(* Logix 5000 project; controller SPONGENT Emulate 5570 rev 30.12; software revision 30.00 *)

TASK MainTask (periodic, rate 500 ms, priority 1, watchdog 500 ms) : MainProgram

MODULES
   Local : Emulate 5570 (ICP 2, rev 30.12)
       : vendor 1 type 0 code 15 (ICP 3, rev 1.1, Output RPI 50 ms)
END_MODULES

VAR_GLOBAL   (* controller tags *)
   SCAN_CYCLE_TIME : DINT := 12;
END_VAR

PROGRAM MainProgram   (* main routine MainRoutine *)
VAR
   Spon_Absorb_i : DINT := 1;
   Spon_BAD_HASHBITLEN : DINT;
   Spon_capacity : DINT := 80;
   Spon_Check_i : DINT := 11;
   Spon_Check_j : DINT := 11;
   Spon_Digest : DINT[256] := ([0] := 211, [1] := 187, [2] := 154, [3] := 14, [4] := 13, [5] := 90, [6] := 242, [7] := 217, [8] := 117, [9] := 72, [10] := 177);
   Spon_DIGESTSIZE : DINT := 88;
   Spon_Hash_i : DINT := 1;
   Spon_Hash_index : DINT;
   Spon_Hash_statrIndex : DINT := 10;
   Spon_hashbitlen : DINT := 88;
   Spon_i : DINT;
   Spon_INV_IV : DINT[512] := ([0] := 63488);
   Spon_IV : DINT[512] := ([0] := 63);
   Spon_j : DINT;
   Spon_Message : DINT[1024] := ([0] := 48, [1] := 48, [2] := 48, [3] := 48, [4] := 48, [5] := 48, [6] := 48, [7] := 48, [8] := 48, [9] := 48, [10] := 48, [11] := 48, [12] := 48, [13] := 48, [14] := 48, [15] := 48, [16] := 48, [17] := 48, [18] := 48, [19] := 48, [20] := 48, [21] := 48, [22] := 48, [23] := 48, [24] := 48, [25] := 48, [26] := 48);
   Spon_messageblock : DINT[1024] := ([0] := 72);
   Spon_MsgBitLen : DINT;
   Spon_nBits : DINT := 88;
   Spon_nRounds : DINT := 45;
   Spon_nSBox : DINT := 11;
   Spon_Pad_bitpos : DINT;
   Spon_Pad_byteind : DINT := 1;
   Spon_Pad_indx : DINT;
   Spon_Permute_i : DINT := 45;
   Spon_Permute_j : DINT := 11;
   Spon_Player_i : DINT := 11;
   Spon_Player_j : DINT := 8;
   Spon_Player_PermutedBitNo : DINT := 87;
   Spon_Player_pos : DINT := 7;
   Spon_Player_tmp : DINT;
   Spon_Player_x : DINT;
   Spon_Player_y : DINT := 10;
   Spon_Player_z : DINT := 87;
   Spon_R_SizeInBytes : DINT := 1;
   Spon_rate : DINT := 8;
   Spon_remainingbitlen : DINT;
   Spon_res : DINT;
   Spon_retnuoCl_lfsr : DINT := 63488;
   Spon_retnuoCl_res : DINT;
   Spon_S : DINT[16] := ([0] := 14, [1] := 13, [2] := 11, [4] := 2, [5] := 1, [6] := 4, [7] := 15, [8] := 7, [9] := 10, [10] := 8, [11] := 5, [12] := 9, [13] := 12, [14] := 3, [15] := 6);
   Spon_SBoxLayer : DINT[256] := ([0] := 238, [1] := 237, [2] := 235, [3] := 224, [4] := 226, [5] := 225, [6] := 228, [7] := 239, [8] := 231, [9] := 234, [10] := 232, [11] := 229, [12] := 233, [13] := 236, [14] := 227, [15] := 230, [16] := 222, [17] := 221, [18] := 219, [19] := 208, [20] := 210, [21] := 209, [22] := 212, [23] := 223, [24] := 215, [25] := 218, [26] := 216, [27] := 213, [28] := 217, [29] := 220, [30] := 211, [31] := 214, [32] := 190, [33] := 189, [34] := 187, [35] := 176, [36] := 178, [37] := 177, [38] := 180, [39] := 191, [40] := 183, [41] := 186, [42] := 184, [43] := 181, [44] := 185, [45] := 188, [46] := 179, [47] := 182, [48] := 14, [49] := 13, [50] := 11, [52] := 2, [53] := 1, [54] := 4, [55] := 15, [56] := 7, [57] := 10, [58] := 8, [59] := 5, [60] := 9,
        [61] := 12, [62] := 3, [63] := 6, [64] := 46, [65] := 45, [66] := 43, [67] := 32, [68] := 34, [69] := 33, [70] := 36, [71] := 47, [72] := 39, [73] := 42, [74] := 40, [75] := 37, [76] := 41, [77] := 44, [78] := 35, [79] := 38, [80] := 30, [81] := 29, [82] := 27, [83] := 16, [84] := 18, [85] := 17, [86] := 20, [87] := 31, [88] := 23, [89] := 26, [90] := 24, [91] := 21, [92] := 25, [93] := 28, [94] := 19, [95] := 22, [96] := 78, [97] := 77, [98] := 75, [99] := 64, [100] := 66, [101] := 65, [102] := 68, [103] := 79, [104] := 71, [105] := 74, [106] := 72, [107] := 69, [108] := 73, [109] := 76, [110] := 67, [111] := 70, [112] := 254, [113] := 253, [114] := 251, [115] := 240, [116] := 242, [117] := 241, [118] := 244, [119] := 255, [120] := 247,
        [121] := 250, [122] := 248, [123] := 245, [124] := 249, [125] := 252, [126] := 243, [127] := 246, [128] := 126, [129] := 125, [130] := 123, [131] := 112, [132] := 114, [133] := 113, [134] := 116, [135] := 127, [136] := 119, [137] := 122, [138] := 120, [139] := 117, [140] := 121, [141] := 124, [142] := 115, [143] := 118, [144] := 174, [145] := 173, [146] := 171, [147] := 160, [148] := 162, [149] := 161, [150] := 164, [151] := 175, [152] := 167, [153] := 170, [154] := 168, [155] := 165, [156] := 169, [157] := 172, [158] := 163, [159] := 166, [160] := 142, [161] := 141, [162] := 139, [163] := 128, [164] := 130, [165] := 129, [166] := 132, [167] := 143, [168] := 135, [169] := 138, [170] := 136, [171] := 133, [172] := 137, [173] := 140, [174] := 131, [175] := 134, [176] := 94, [177] := 93, [178] := 91, [179] := 80, [180] := 82,
        [181] := 81, [182] := 84, [183] := 95, [184] := 87, [185] := 90, [186] := 88, [187] := 85, [188] := 89, [189] := 92, [190] := 83, [191] := 86, [192] := 158, [193] := 157, [194] := 155, [195] := 144, [196] := 146, [197] := 145, [198] := 148, [199] := 159, [200] := 151, [201] := 154, [202] := 152, [203] := 149, [204] := 153, [205] := 156, [206] := 147, [207] := 150, [208] := 206, [209] := 205, [210] := 203, [211] := 192, [212] := 194, [213] := 193, [214] := 196, [215] := 207, [216] := 199, [217] := 202, [218] := 200, [219] := 197, [220] := 201, [221] := 204, [222] := 195, [223] := 198, [224] := 62, [225] := 61, [226] := 59, [227] := 48, [228] := 50, [229] := 49, [230] := 52, [231] := 63, [232] := 55, [233] := 58, [234] := 56, [235] := 53, [236] := 57, [237] := 60, [238] := 51, [239] := 54, [240] := 110,
        [241] := 109, [242] := 107, [243] := 96, [244] := 98, [245] := 97, [246] := 100, [247] := 111, [248] := 103, [249] := 106, [250] := 104, [251] := 101, [252] := 105, [253] := 108, [254] := 99, [255] := 102);
   Spon_Slayer_input : DINT := 241;
   Spon_Slayer_res : DINT;
   Spon_Squeeze_i : DINT := 1;
   Spon_State : DINT[256] := ([0] := 177, [1] := 249, [2] := 148, [3] := 195, [4] := 111, [5] := 169, [6] := 251, [7] := 236, [8] := 167, [9] := 175, [10] := 126);
   Spon_State_tmp : DINT[256] := ([0] := 177, [1] := 249, [2] := 148, [3] := 195, [4] := 111, [5] := 169, [6] := 251, [7] := 236, [8] := 167, [9] := 175, [10] := 126);
   Spon_SUCCESS : DINT;
   Spon_Ver : DINT := 88808;
   Test_i : DINT := 27;
END_VAR

ROUTINE MainRoutine   (* ladder *)
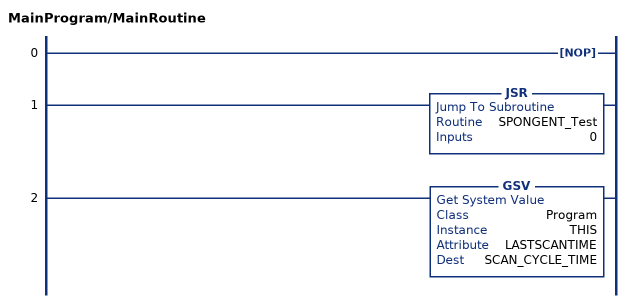
   0: NOP();
   1: JSR(SPONGENT_Test,0);
   2: GSV(Program,THIS,LASTSCANTIME,SCAN_CYCLE_TIME);
END_ROUTINE

ROUTINE SPONGENT   (* structured text *)
   JSR(SPONGENT_Init);
   
   
   
   //Spon_hashval, state
   
   
   
   
   /* Absorb available message blocks */
   Spon_Hash_statrIndex:=0;
   While Spon_MsgBitLen >= Spon_rate do
   	//memcpy(state.messageblock, data, R_SizeInBytes);
   	for Spon_Hash_i:=0 to Spon_R_SizeInBytes-1 by 1 do
   		Spon_messageblock[Spon_Hash_i]:=Spon_Message[Spon_Hash_statrIndex+Spon_Hash_i];
   	end_for;
   
   
   	JSR(SPONGENT_Absorb);
   	Spon_MsgBitLen:=Spon_MsgBitLen-Spon_rate;
   	Spon_Hash_statrIndex:=Spon_Hash_statrIndex+Spon_R_SizeInBytes;
   
   end_while;
   
   
   
   //databitlen/8 + (databitlen%8?1:0)
   Spon_Hash_index:=Spon_MsgBitLen mod 8;
   if Spon_Hash_index=0 then
   	Spon_Hash_index:=Spon_MsgBitLen / 8;
   else
   	Spon_Hash_index:=Spon_MsgBitLen / 8 + 1;
   end_if;
   
   if Spon_MsgBitLen>0 then
   //memcpy(state.messageblock, data, databitlen/8 + (databitlen%8?1:0));
   	for Spon_Hash_i:=0 to Spon_Hash_index-1 by 1 do
   		Spon_messageblock[Spon_Hash_i]:=Spon_Message[Spon_Hash_statrIndex+Spon_Hash_i];
   	end_for;
   	Spon_remainingbitlen:=Spon_MsgBitLen;
   else
   	for Spon_Hash_i:=0 to Spon_R_SizeInBytes-1 by 1 do
   		Spon_messageblock[Spon_Hash_i]:=0;
   	end_for;
   	Spon_remainingbitlen:=Spon_MsgBitLen;
   end_if;
   
   
   JSR(SPONGENT_Pad);
   
   JSR(SPONGENT_Absorb);
   Spon_hashbitlen:=Spon_hashbitlen+Spon_rate;
   
   /* Squeeze data blocks */
   Spon_Hash_statrIndex:=0;
   while Spon_hashbitlen<Spon_DIGESTSIZE do
   	JSR(SPONGENT_Squeeze);
   
   
   	for Spon_Hash_i:=0 to Spon_R_SizeInBytes-1 by 1 do
   		Spon_Digest[Spon_Hash_statrIndex+Spon_Hash_i]:=Spon_messageblock[Spon_Hash_i];
   	end_for;
   
   	Spon_hashbitlen:=Spon_hashbitlen+Spon_rate;
   	Spon_Hash_statrIndex:=Spon_Hash_statrIndex+Spon_R_SizeInBytes;
   
   end_while;
   
   
   
   for Spon_Hash_i:=0 to Spon_R_SizeInBytes-1 by 1 do
   	Spon_Digest[Spon_Hash_statrIndex+Spon_Hash_i]:=Spon_State[Spon_Hash_i];
   end_for;
   
   
   
   
   
   
   
   
   
   
   
   
   
END_ROUTINE

ROUTINE SPONGENT_Absorb   (* structured text *)
   (*
   int i;
   	for(i = 0; i < R_SizeInBytes; i++)
   		state->value[i] ^= state->messageblock[i];
    	Permute(state);
   
   	return SUCCESS;
   
   	*)
   
   For Spon_Absorb_i:=0 to Spon_R_SizeInBytes-1 by 1 Do
   	Spon_State[Spon_Absorb_i]:= Spon_State[Spon_Absorb_i] Xor Spon_messageblock[Spon_Absorb_i];
   End_for;
   
   JSR(SPONGENT_Permute);
END_ROUTINE

ROUTINE SPONGENT_Init   (* structured text *)
   	Spon_INV_IV[0]:=25344;
   	Spon_INV_IV[1]:=22528;
   	Spon_INV_IV[2]:=38400;
   	Spon_INV_IV[3]:=42240;
   	Spon_INV_IV[4]:=26880;
   	Spon_INV_IV[5]:=6656;
   	Spon_INV_IV[6]:=17920;
   	Spon_INV_IV[7]:=37120;
   	Spon_INV_IV[8]:=41984;
   	Spon_INV_IV[9]:=26880;
   	Spon_INV_IV[10]:=6656;
   	Spon_INV_IV[11]:=17920;
   	Spon_INV_IV[12]:=37120;
   	Spon_INV_IV[13]:=41984;
   	Spon_INV_IV[14]:=26880;
   	Spon_INV_IV[15]:=6656;
   	Spon_INV_IV[16]:=17920;
   	Spon_INV_IV[17]:=37120;
   	Spon_INV_IV[18]:=41984;
   	Spon_INV_IV[19]:=26880;
   	Spon_INV_IV[20]:=6656;
   	Spon_INV_IV[21]:=17920;
   	Spon_INV_IV[22]:=37120;
   	Spon_INV_IV[23]:=41984;
   	Spon_INV_IV[24]:=26880;
   	Spon_INV_IV[25]:=6656;
   	Spon_INV_IV[26]:=17920;
   	Spon_INV_IV[27]:=37120;
   	Spon_INV_IV[28]:=41984;
   	Spon_INV_IV[29]:=26880;
   	Spon_INV_IV[30]:=6656;
   	Spon_INV_IV[31]:=17920;
   	Spon_INV_IV[32]:=37120;
   	Spon_INV_IV[33]:=41984;
   	Spon_INV_IV[34]:=26880;
   	Spon_INV_IV[35]:=6656;
   	Spon_INV_IV[36]:=17920;
   	Spon_INV_IV[37]:=37120;
   	Spon_INV_IV[38]:=41984;
   	Spon_INV_IV[39]:=26880;
   	Spon_INV_IV[40]:=6656;
   	Spon_INV_IV[41]:=17920;
   	Spon_INV_IV[42]:=37120;
   	Spon_INV_IV[43]:=41984;
   	Spon_INV_IV[44]:=26880;
   	Spon_INV_IV[45]:=6656;
   	Spon_INV_IV[46]:=17920;
   	Spon_INV_IV[47]:=37120;
   	Spon_INV_IV[48]:=41984;
   	Spon_INV_IV[49]:=26880;
   	Spon_INV_IV[50]:=6656;
   	Spon_INV_IV[51]:=17920;
   	Spon_INV_IV[52]:=37120;
   	Spon_INV_IV[53]:=41984;
   	Spon_INV_IV[54]:=26880;
   	Spon_INV_IV[55]:=6656;
   	Spon_INV_IV[56]:=17920;
   	Spon_INV_IV[57]:=37120;
   	Spon_INV_IV[58]:=41984;
   	Spon_INV_IV[59]:=26880;
   	Spon_INV_IV[60]:=6656;
   	Spon_INV_IV[61]:=17920;
   	Spon_INV_IV[62]:=37120;
   	Spon_INV_IV[63]:=41984;
   	Spon_INV_IV[64]:=26880;
   	Spon_INV_IV[65]:=6656;
   	Spon_INV_IV[66]:=17920;
   	Spon_INV_IV[67]:=37120;
   	Spon_INV_IV[68]:=41984;
   	Spon_INV_IV[69]:=26880;
   	Spon_INV_IV[70]:=6656;
   	Spon_INV_IV[71]:=17920;
   	Spon_INV_IV[72]:=37120;
   	Spon_INV_IV[73]:=41984;
   	Spon_INV_IV[74]:=26880;
   	Spon_INV_IV[75]:=6656;
   	Spon_INV_IV[76]:=17920;
   	Spon_INV_IV[77]:=37120;
   	Spon_INV_IV[78]:=41984;
   	Spon_INV_IV[79]:=26880;
   	Spon_INV_IV[80]:=6656;
   	Spon_INV_IV[81]:=17920;
   	Spon_INV_IV[82]:=37120;
   	Spon_INV_IV[83]:=41984;
   	Spon_INV_IV[84]:=26880;
   	Spon_INV_IV[85]:=6656;
   	Spon_INV_IV[86]:=17920;
   	Spon_INV_IV[87]:=37120;
   	Spon_INV_IV[88]:=41984;
   	Spon_INV_IV[89]:=26880;
   	Spon_INV_IV[90]:=6656;
   	Spon_INV_IV[91]:=17920;
   	Spon_INV_IV[92]:=37120;
   	Spon_INV_IV[93]:=41984;
   	Spon_INV_IV[94]:=26880;
   	Spon_INV_IV[95]:=6656;
   	Spon_INV_IV[96]:=17920;
   	Spon_INV_IV[97]:=37120;
   	Spon_INV_IV[98]:=41984;
   	Spon_INV_IV[99]:=26880;
   	Spon_INV_IV[100]:=6656;
   	Spon_INV_IV[101]:=17920;
   	Spon_INV_IV[102]:=37120;
   	Spon_INV_IV[103]:=41984;
   	Spon_INV_IV[104]:=26880;
   	Spon_INV_IV[105]:=6656;
   	Spon_INV_IV[106]:=17920;
   	Spon_INV_IV[107]:=37120;
   	Spon_INV_IV[108]:=41984;
   	Spon_INV_IV[109]:=26880;
   	Spon_INV_IV[110]:=6656;
   	Spon_INV_IV[111]:=17920;
   	Spon_INV_IV[112]:=37120;
   	Spon_INV_IV[113]:=41984;
   	Spon_INV_IV[114]:=26880;
   	Spon_INV_IV[115]:=6656;
   	Spon_INV_IV[116]:=17920;
   	Spon_INV_IV[117]:=37120;
   	Spon_INV_IV[118]:=41984;
   	Spon_INV_IV[119]:=26880;
   	Spon_INV_IV[120]:=6656;
   	Spon_INV_IV[121]:=17920;
   	Spon_INV_IV[122]:=37120;
   	Spon_INV_IV[123]:=41984;
   	Spon_INV_IV[124]:=26880;
   	Spon_INV_IV[125]:=6656;
   	Spon_INV_IV[126]:=17920;
   	Spon_INV_IV[127]:=37120;
   	Spon_INV_IV[128]:=41984;
   	Spon_INV_IV[129]:=26880;
   	Spon_INV_IV[130]:=6656;
   	Spon_INV_IV[131]:=17920;
   	Spon_INV_IV[132]:=37120;
   	Spon_INV_IV[133]:=41984;
   	Spon_INV_IV[134]:=26880;
   
   
   	Spon_IV[0]:=198;
   	Spon_IV[1]:=26;
   	Spon_IV[2]:=105;
   	Spon_IV[3]:=165;
   	Spon_IV[4]:=150;
   	Spon_IV[5]:=88;
   	Spon_IV[6]:=98;
   	Spon_IV[7]:=137;
   	Spon_IV[8]:=37;
   	Spon_IV[9]:=150;
   	Spon_IV[10]:=88;
   	Spon_IV[11]:=98;
   	Spon_IV[12]:=137;
   	Spon_IV[13]:=37;
   	Spon_IV[14]:=150;
   	Spon_IV[15]:=88;
   	Spon_IV[16]:=98;
   	Spon_IV[17]:=137;
   	Spon_IV[18]:=37;
   	Spon_IV[19]:=150;
   	Spon_IV[20]:=88;
   	Spon_IV[21]:=98;
   	Spon_IV[22]:=137;
   	Spon_IV[23]:=37;
   	Spon_IV[24]:=150;
   	Spon_IV[25]:=88;
   	Spon_IV[26]:=98;
   	Spon_IV[27]:=137;
   	Spon_IV[28]:=37;
   	Spon_IV[29]:=150;
   	Spon_IV[30]:=88;
   	Spon_IV[31]:=98;
   	Spon_IV[32]:=137;
   	Spon_IV[33]:=37;
   	Spon_IV[34]:=150;
   	Spon_IV[35]:=88;
   	Spon_IV[36]:=98;
   	Spon_IV[37]:=137;
   	Spon_IV[38]:=37;
   	Spon_IV[39]:=150;
   	Spon_IV[40]:=88;
   	Spon_IV[41]:=98;
   	Spon_IV[42]:=137;
   	Spon_IV[43]:=37;
   	Spon_IV[44]:=150;
   	Spon_IV[45]:=88;
   	Spon_IV[46]:=98;
   	Spon_IV[47]:=137;
   	Spon_IV[48]:=37;
   	Spon_IV[49]:=150;
   	Spon_IV[50]:=88;
   	Spon_IV[51]:=98;
   	Spon_IV[52]:=137;
   	Spon_IV[53]:=37;
   	Spon_IV[54]:=150;
   	Spon_IV[55]:=88;
   	Spon_IV[56]:=98;
   	Spon_IV[57]:=137;
   	Spon_IV[58]:=37;
   	Spon_IV[59]:=150;
   	Spon_IV[60]:=88;
   	Spon_IV[61]:=98;
   	Spon_IV[62]:=137;
   	Spon_IV[63]:=37;
   	Spon_IV[64]:=150;
   	Spon_IV[65]:=88;
   	Spon_IV[66]:=98;
   	Spon_IV[67]:=137;
   	Spon_IV[68]:=37;
   	Spon_IV[69]:=150;
   	Spon_IV[70]:=88;
   	Spon_IV[71]:=98;
   	Spon_IV[72]:=137;
   	Spon_IV[73]:=37;
   	Spon_IV[74]:=150;
   	Spon_IV[75]:=88;
   	Spon_IV[76]:=98;
   	Spon_IV[77]:=137;
   	Spon_IV[78]:=37;
   	Spon_IV[79]:=150;
   	Spon_IV[80]:=88;
   	Spon_IV[81]:=98;
   	Spon_IV[82]:=137;
   	Spon_IV[83]:=37;
   	Spon_IV[84]:=150;
   	Spon_IV[85]:=88;
   	Spon_IV[86]:=98;
   	Spon_IV[87]:=137;
   	Spon_IV[88]:=37;
   	Spon_IV[89]:=150;
   	Spon_IV[90]:=88;
   	Spon_IV[91]:=98;
   	Spon_IV[92]:=137;
   	Spon_IV[93]:=37;
   	Spon_IV[94]:=150;
   	Spon_IV[95]:=88;
   	Spon_IV[96]:=98;
   	Spon_IV[97]:=137;
   	Spon_IV[98]:=37;
   	Spon_IV[99]:=150;
   	Spon_IV[100]:=88;
   	Spon_IV[101]:=98;
   	Spon_IV[102]:=137;
   	Spon_IV[103]:=37;
   	Spon_IV[104]:=150;
   	Spon_IV[105]:=88;
   	Spon_IV[106]:=98;
   	Spon_IV[107]:=137;
   	Spon_IV[108]:=37;
   	Spon_IV[109]:=150;
   	Spon_IV[110]:=88;
   	Spon_IV[111]:=98;
   	Spon_IV[112]:=137;
   	Spon_IV[113]:=37;
   	Spon_IV[114]:=150;
   	Spon_IV[115]:=88;
   	Spon_IV[116]:=98;
   	Spon_IV[117]:=137;
   	Spon_IV[118]:=37;
   	Spon_IV[119]:=150;
   	Spon_IV[120]:=88;
   	Spon_IV[121]:=98;
   	Spon_IV[122]:=137;
   	Spon_IV[123]:=37;
   	Spon_IV[124]:=150;
   	Spon_IV[125]:=88;
   	Spon_IV[126]:=98;
   	Spon_IV[127]:=137;
   	Spon_IV[128]:=37;
   	Spon_IV[129]:=150;
   	Spon_IV[130]:=88;
   	Spon_IV[131]:=98;
   	Spon_IV[132]:=137;
   	Spon_IV[133]:=37;
   	Spon_IV[134]:=150;
   	Spon_IV[135]:=88;
   
   
   		Spon_SBoxLayer[0]:=238;
   		Spon_SBoxLayer[1]:=237;
   		Spon_SBoxLayer[2]:=235;
   		Spon_SBoxLayer[3]:=224;
   		Spon_SBoxLayer[4]:=226;
   		Spon_SBoxLayer[5]:=225;
   		Spon_SBoxLayer[6]:=228;
   		Spon_SBoxLayer[7]:=239;
   		Spon_SBoxLayer[8]:=231;
   		Spon_SBoxLayer[9]:=234;
   		Spon_SBoxLayer[10]:=232;
   		Spon_SBoxLayer[11]:=229;
   		Spon_SBoxLayer[12]:=233;
   		Spon_SBoxLayer[13]:=236;
   		Spon_SBoxLayer[14]:=227;
   		Spon_SBoxLayer[15]:=230;
   		Spon_SBoxLayer[16]:=222;
   		Spon_SBoxLayer[17]:=221;
   		Spon_SBoxLayer[18]:=219;
   		Spon_SBoxLayer[19]:=208;
   		Spon_SBoxLayer[20]:=210;
   		Spon_SBoxLayer[21]:=209;
   		Spon_SBoxLayer[22]:=212;
   		Spon_SBoxLayer[23]:=223;
   		Spon_SBoxLayer[24]:=215;
   		Spon_SBoxLayer[25]:=218;
   		Spon_SBoxLayer[26]:=216;
   		Spon_SBoxLayer[27]:=213;
   		Spon_SBoxLayer[28]:=217;
   		Spon_SBoxLayer[29]:=220;
   		Spon_SBoxLayer[30]:=211;
   		Spon_SBoxLayer[31]:=214;
   		Spon_SBoxLayer[32]:=190;
   		Spon_SBoxLayer[33]:=189;
   		Spon_SBoxLayer[34]:=187;
   		Spon_SBoxLayer[35]:=176;
   		Spon_SBoxLayer[36]:=178;
   		Spon_SBoxLayer[37]:=177;
   		Spon_SBoxLayer[38]:=180;
   		Spon_SBoxLayer[39]:=191;
   		Spon_SBoxLayer[40]:=183;
   		Spon_SBoxLayer[41]:=186;
   		Spon_SBoxLayer[42]:=184;
   		Spon_SBoxLayer[43]:=181;
   		Spon_SBoxLayer[44]:=185;
   		Spon_SBoxLayer[45]:=188;
   		Spon_SBoxLayer[46]:=179;
   		Spon_SBoxLayer[47]:=182;
   		Spon_SBoxLayer[48]:=14;
   		Spon_SBoxLayer[49]:=13;
   		Spon_SBoxLayer[50]:=11;
   		Spon_SBoxLayer[51]:=0;
   		Spon_SBoxLayer[52]:=2;
   		Spon_SBoxLayer[53]:=1;
   		Spon_SBoxLayer[54]:=4;
   		Spon_SBoxLayer[55]:=15;
   		Spon_SBoxLayer[56]:=7;
   		Spon_SBoxLayer[57]:=10;
   		Spon_SBoxLayer[58]:=8;
   		Spon_SBoxLayer[59]:=5;
   		Spon_SBoxLayer[60]:=9;
   		Spon_SBoxLayer[61]:=12;
   		Spon_SBoxLayer[62]:=3;
   		Spon_SBoxLayer[63]:=6;
   		Spon_SBoxLayer[64]:=46;
   		Spon_SBoxLayer[65]:=45;
   		Spon_SBoxLayer[66]:=43;
   		Spon_SBoxLayer[67]:=32;
   		Spon_SBoxLayer[68]:=34;
   		Spon_SBoxLayer[69]:=33;
   		Spon_SBoxLayer[70]:=36;
   		Spon_SBoxLayer[71]:=47;
   		Spon_SBoxLayer[72]:=39;
   		Spon_SBoxLayer[73]:=42;
   		Spon_SBoxLayer[74]:=40;
   		Spon_SBoxLayer[75]:=37;
   		Spon_SBoxLayer[76]:=41;
   		Spon_SBoxLayer[77]:=44;
   		Spon_SBoxLayer[78]:=35;
   		Spon_SBoxLayer[79]:=38;
   		Spon_SBoxLayer[80]:=30;
   		Spon_SBoxLayer[81]:=29;
   		Spon_SBoxLayer[82]:=27;
   		Spon_SBoxLayer[83]:=16;
   		Spon_SBoxLayer[84]:=18;
   		Spon_SBoxLayer[85]:=17;
   		Spon_SBoxLayer[86]:=20;
   		Spon_SBoxLayer[87]:=31;
   		Spon_SBoxLayer[88]:=23;
   		Spon_SBoxLayer[89]:=26;
   		Spon_SBoxLayer[90]:=24;
   		Spon_SBoxLayer[91]:=21;
   		Spon_SBoxLayer[92]:=25;
   		Spon_SBoxLayer[93]:=28;
   		Spon_SBoxLayer[94]:=19;
   		Spon_SBoxLayer[95]:=22;
   		Spon_SBoxLayer[96]:=78;
   		Spon_SBoxLayer[97]:=77;
   		Spon_SBoxLayer[98]:=75;
   		Spon_SBoxLayer[99]:=64;
   		Spon_SBoxLayer[100]:=66;
   		Spon_SBoxLayer[101]:=65;
   		Spon_SBoxLayer[102]:=68;
   		Spon_SBoxLayer[103]:=79;
   		Spon_SBoxLayer[104]:=71;
   		Spon_SBoxLayer[105]:=74;
   		Spon_SBoxLayer[106]:=72;
   		Spon_SBoxLayer[107]:=69;
   		Spon_SBoxLayer[108]:=73;
   		Spon_SBoxLayer[109]:=76;
   		Spon_SBoxLayer[110]:=67;
   		Spon_SBoxLayer[111]:=70;
   		Spon_SBoxLayer[112]:=254;
   		Spon_SBoxLayer[113]:=253;
   		Spon_SBoxLayer[114]:=251;
   		Spon_SBoxLayer[115]:=240;
   		Spon_SBoxLayer[116]:=242;
   		Spon_SBoxLayer[117]:=241;
   		Spon_SBoxLayer[118]:=244;
   		Spon_SBoxLayer[119]:=255;
   		Spon_SBoxLayer[120]:=247;
   		Spon_SBoxLayer[121]:=250;
   		Spon_SBoxLayer[122]:=248;
   		Spon_SBoxLayer[123]:=245;
   		Spon_SBoxLayer[124]:=249;
   		Spon_SBoxLayer[125]:=252;
   		Spon_SBoxLayer[126]:=243;
   		Spon_SBoxLayer[127]:=246;
   		Spon_SBoxLayer[128]:=126;
   		Spon_SBoxLayer[129]:=125;
   		Spon_SBoxLayer[130]:=123;
   		Spon_SBoxLayer[131]:=112;
   		Spon_SBoxLayer[132]:=114;
   		Spon_SBoxLayer[133]:=113;
   		Spon_SBoxLayer[134]:=116;
   		Spon_SBoxLayer[135]:=127;
   		Spon_SBoxLayer[136]:=119;
   		Spon_SBoxLayer[137]:=122;
   		Spon_SBoxLayer[138]:=120;
   		Spon_SBoxLayer[139]:=117;
   		Spon_SBoxLayer[140]:=121;
   		Spon_SBoxLayer[141]:=124;
   		Spon_SBoxLayer[142]:=115;
   		Spon_SBoxLayer[143]:=118;
   		Spon_SBoxLayer[144]:=174;
   		Spon_SBoxLayer[145]:=173;
   		Spon_SBoxLayer[146]:=171;
   		Spon_SBoxLayer[147]:=160;
   		Spon_SBoxLayer[148]:=162;
   		Spon_SBoxLayer[149]:=161;
   		Spon_SBoxLayer[150]:=164;
   		Spon_SBoxLayer[151]:=175;
   		Spon_SBoxLayer[152]:=167;
   		Spon_SBoxLayer[153]:=170;
   		Spon_SBoxLayer[154]:=168;
   		Spon_SBoxLayer[155]:=165;
   		Spon_SBoxLayer[156]:=169;
   		Spon_SBoxLayer[157]:=172;
   		Spon_SBoxLayer[158]:=163;
   		Spon_SBoxLayer[159]:=166;
   		Spon_SBoxLayer[160]:=142;
   		Spon_SBoxLayer[161]:=141;
   		Spon_SBoxLayer[162]:=139;
   		Spon_SBoxLayer[163]:=128;
   		Spon_SBoxLayer[164]:=130;
   		Spon_SBoxLayer[165]:=129;
   		Spon_SBoxLayer[166]:=132;
   		Spon_SBoxLayer[167]:=143;
   		Spon_SBoxLayer[168]:=135;
   		Spon_SBoxLayer[169]:=138;
   		Spon_SBoxLayer[170]:=136;
   		Spon_SBoxLayer[171]:=133;
   		Spon_SBoxLayer[172]:=137;
   		Spon_SBoxLayer[173]:=140;
   		Spon_SBoxLayer[174]:=131;
   		Spon_SBoxLayer[175]:=134;
   		Spon_SBoxLayer[176]:=94;
   		Spon_SBoxLayer[177]:=93;
   		Spon_SBoxLayer[178]:=91;
   		Spon_SBoxLayer[179]:=80;
   		Spon_SBoxLayer[180]:=82;
   		Spon_SBoxLayer[181]:=81;
   		Spon_SBoxLayer[182]:=84;
   		Spon_SBoxLayer[183]:=95;
   		Spon_SBoxLayer[184]:=87;
   		Spon_SBoxLayer[185]:=90;
   		Spon_SBoxLayer[186]:=88;
   		Spon_SBoxLayer[187]:=85;
   		Spon_SBoxLayer[188]:=89;
   		Spon_SBoxLayer[189]:=92;
   		Spon_SBoxLayer[190]:=83;
   		Spon_SBoxLayer[191]:=86;
   		Spon_SBoxLayer[192]:=158;
   		Spon_SBoxLayer[193]:=157;
   		Spon_SBoxLayer[194]:=155;
   		Spon_SBoxLayer[195]:=144;
   		Spon_SBoxLayer[196]:=146;
   		Spon_SBoxLayer[197]:=145;
   		Spon_SBoxLayer[198]:=148;
   		Spon_SBoxLayer[199]:=159;
   		Spon_SBoxLayer[200]:=151;
   		Spon_SBoxLayer[201]:=154;
   		Spon_SBoxLayer[202]:=152;
   		Spon_SBoxLayer[203]:=149;
   		Spon_SBoxLayer[204]:=153;
   		Spon_SBoxLayer[205]:=156;
   		Spon_SBoxLayer[206]:=147;
   		Spon_SBoxLayer[207]:=150;
   		Spon_SBoxLayer[208]:=206;
   		Spon_SBoxLayer[209]:=205;
   		Spon_SBoxLayer[210]:=203;
   		Spon_SBoxLayer[211]:=192;
   		Spon_SBoxLayer[212]:=194;
   		Spon_SBoxLayer[213]:=193;
   		Spon_SBoxLayer[214]:=196;
   		Spon_SBoxLayer[215]:=207;
   		Spon_SBoxLayer[216]:=199;
   		Spon_SBoxLayer[217]:=202;
   		Spon_SBoxLayer[218]:=200;
   		Spon_SBoxLayer[219]:=197;
   		Spon_SBoxLayer[220]:=201;
   		Spon_SBoxLayer[221]:=204;
   		Spon_SBoxLayer[222]:=195;
   		Spon_SBoxLayer[223]:=198;
   		Spon_SBoxLayer[224]:=62;
   		Spon_SBoxLayer[225]:=61;
   		Spon_SBoxLayer[226]:=59;
   		Spon_SBoxLayer[227]:=48;
   		Spon_SBoxLayer[228]:=50;
   		Spon_SBoxLayer[229]:=49;
   		Spon_SBoxLayer[230]:=52;
   		Spon_SBoxLayer[231]:=63;
   		Spon_SBoxLayer[232]:=55;
   		Spon_SBoxLayer[233]:=58;
   		Spon_SBoxLayer[234]:=56;
   		Spon_SBoxLayer[235]:=53;
   		Spon_SBoxLayer[236]:=57;
   		Spon_SBoxLayer[237]:=60;
   		Spon_SBoxLayer[238]:=51;
   		Spon_SBoxLayer[239]:=54;
   		Spon_SBoxLayer[240]:=110;
   		Spon_SBoxLayer[241]:=109;
   		Spon_SBoxLayer[242]:=107;
   		Spon_SBoxLayer[243]:=96;
   		Spon_SBoxLayer[244]:=98;
   		Spon_SBoxLayer[245]:=97;
   		Spon_SBoxLayer[246]:=100;
   		Spon_SBoxLayer[247]:=111;
   		Spon_SBoxLayer[248]:=103;
   		Spon_SBoxLayer[249]:=106;
   		Spon_SBoxLayer[250]:=104;
   		Spon_SBoxLayer[251]:=101;
   		Spon_SBoxLayer[252]:=105;
   		Spon_SBoxLayer[253]:=108;
   		Spon_SBoxLayer[254]:=99;
   		Spon_SBoxLayer[255]:=102;
   CASE Spon_Ver OF
   	 88808:
   		Spon_rate:=8;
   		Spon_capacity:=80;
   		Spon_DIGESTSIZE:=88;
   		Spon_nRounds:=45;
   
   		Spon_R_SizeInBytes:=1;
   		Spon_nBits:=88;
   		Spon_nSBox:=11;
   	 8817688:
   		Spon_rate:=88;
   		Spon_capacity:=176;
   		Spon_DIGESTSIZE:=88;
   		Spon_nRounds:=135;
   		Spon_R_SizeInBytes:=11;
   		Spon_nBits:=264;
   		Spon_nSBox:=33;
   	 1281288:
   		Spon_rate:=8;
   		Spon_capacity:=128;
   		Spon_DIGESTSIZE:=128;
   		Spon_nRounds:=70;
   		Spon_R_SizeInBytes:=1;
   		Spon_nBits:=136;
   		Spon_nSBox:=17;
   	 128256128:
   		Spon_rate:=128;
   		Spon_capacity:=256;
   		Spon_DIGESTSIZE:=128;
   		Spon_nRounds:=195;
   		Spon_R_SizeInBytes:=16;
   		Spon_nBits:=384;
   		Spon_nSBox:=48;
   	 16016016:
   		Spon_rate:=16;
   		Spon_capacity:=160;
   		Spon_DIGESTSIZE:=160;
   		Spon_nRounds:=90;
   		Spon_R_SizeInBytes:=2;
   		Spon_nBits:=176;
   		Spon_nSBox:=22;
   	 16016080:
   		Spon_rate:=80;
   		Spon_capacity:=160;
   		Spon_DIGESTSIZE:=160;
   		Spon_nRounds:=120;
   		Spon_R_SizeInBytes:=10;
   		Spon_nBits:=240;
   		Spon_nSBox:=30;
   	 160320160:
   		Spon_rate:=160;
   		Spon_capacity:=320;
   		Spon_DIGESTSIZE:=160;
   		Spon_nRounds:=240;
   		Spon_R_SizeInBytes:=20;
   		Spon_nBits:=480;
   		Spon_nSBox:=60;
   	 22422416:
   		Spon_rate:=16;
   		Spon_capacity:=224;
   		Spon_DIGESTSIZE:=224;
   		Spon_nRounds:=120;
   		Spon_R_SizeInBytes:=2;
   		Spon_nBits:=240;
   		Spon_nSBox:=30;
   	 224224112:
   		Spon_rate:=112;
   		Spon_capacity:=224;
   		Spon_DIGESTSIZE:=224;
   		Spon_nRounds:=170;
   		Spon_R_SizeInBytes:=14;
   		Spon_nBits:=336;
   		Spon_nSBox:=42;
   	 224448224:
   		Spon_rate:=224;
   		Spon_capacity:=448;
   		Spon_DIGESTSIZE:=224;
   		Spon_nRounds:=340;
   		Spon_R_SizeInBytes:=28;
   		Spon_nBits:=672;
   		Spon_nSBox:=84;
   	 25625616:
   		Spon_rate:=16;
   		Spon_capacity:=256;
   		Spon_DIGESTSIZE:=256;
   		Spon_nRounds:=140;
   		Spon_R_SizeInBytes:=2;
   		Spon_nBits:=272;
   		Spon_nSBox:=34;
   	 256256128:
   		Spon_rate:=128;
   		Spon_capacity:=256;
   		Spon_DIGESTSIZE:=256;
   		Spon_nRounds:=195;
   		Spon_R_SizeInBytes:=16;
   		Spon_nBits:=384;
   		Spon_nSBox:=48;
   	 256512256:
   		Spon_rate:=256;
   		Spon_capacity:=512;
   		Spon_DIGESTSIZE:=256;
   		Spon_nRounds:=385;
   		Spon_R_SizeInBytes:=32;
   		Spon_nBits:=768;
   		Spon_nSBox:=96;
   End_CASE;
   
   
   
   
   
   
   
   for Spon_Check_i:=0 to Spon_nSBox-1 by 1 do
   	Spon_State[Spon_Check_i]:=0;
   end_for;
   
   Spon_hashbitlen:=0;
   
   
   Spon_Check_j:=Spon_DIGESTSIZE/8;
   for Spon_Check_i:=0 to Spon_Check_j-1 by 1 do
   	Spon_Digest[Spon_Check_i]:=0;
   end_for;
END_ROUTINE

ROUTINE SPONGENT_Pad   (* structured text *)
   (*
   HashReturn Pad(hashState *state)
   {
           int byteind = state->remainingbitlen/8; /* byte index of remaining byte */
           int bitpos = state->remainingbitlen%8; /* bit position in last byte */
   
           /* make unoccupied bits 0 */
           if(bitpos)
                   state->messageblock[byteind] &= 0xFF<<(8-bitpos);
   
           /* add single 1-bit */
           if(bitpos){
                   state->messageblock[byteind] |= 0x80>>(bitpos);}
           else{
                   state->messageblock[byteind] = 0x80;}
   
           /* add 0-bits until we have rate bits */
           while(byteind!=R_SizeInBytes)
           {
                   byteind++;
                   state->messageblock[byteind] = 0;
           }
           return SUCCESS;
   }
   
   *)
   	Spon_Pad_byteind:= Spon_remainingbitlen/8;
   	Spon_Pad_bitpos:= Spon_remainingbitlen mod 8;
   	if Spon_Pad_bitpos<> 0 then
   		Spon_Pad_indx:= 8-Spon_Pad_bitpos;
   		Case Spon_Pad_indx of
   			1:
   				Spon_messageblock[Spon_Pad_byteind]:= Spon_messageblock[Spon_Pad_byteind] and 16#1fe;
   			2:
   				Spon_messageblock[Spon_Pad_byteind]:= Spon_messageblock[Spon_Pad_byteind] and 16#3fc;
   			3:
   				Spon_messageblock[Spon_Pad_byteind]:= Spon_messageblock[Spon_Pad_byteind] and 16#7fb;
   			4:
   				Spon_messageblock[Spon_Pad_byteind]:= Spon_messageblock[Spon_Pad_byteind] and 16#FF0;
   			5:
   				Spon_messageblock[Spon_Pad_byteind]:= Spon_messageblock[Spon_Pad_byteind] and 16#1fe0;
   			6:
   				Spon_messageblock[Spon_Pad_byteind]:= Spon_messageblock[Spon_Pad_byteind] and 16#3fc0;
   			7:
   				Spon_messageblock[Spon_Pad_byteind]:= Spon_messageblock[Spon_Pad_byteind] and 16#7F80;
   			8:
   				Spon_messageblock[Spon_Pad_byteind]:= Spon_messageblock[Spon_Pad_byteind] and 16#FF00;
   		End_case;
   
   	End_if;
   
   
   	if Spon_Pad_bitpos<> 0 then
   
   		Case Spon_Pad_bitpos of
   			0:Spon_messageblock[Spon_Pad_byteind]:= Spon_messageblock[Spon_Pad_byteind] or 128;
   			1: Spon_messageblock[Spon_Pad_byteind]:= Spon_messageblock[Spon_Pad_byteind] or 64;
   			2: Spon_messageblock[Spon_Pad_byteind]:= Spon_messageblock[Spon_Pad_byteind] or 32;
   			3:
   				Spon_messageblock[Spon_Pad_byteind]:= Spon_messageblock[Spon_Pad_byteind] or 16;
   			4:
   				Spon_messageblock[Spon_Pad_byteind]:= Spon_messageblock[Spon_Pad_byteind] or 16#8;
   			5:
   				Spon_messageblock[Spon_Pad_byteind]:= Spon_messageblock[Spon_Pad_byteind] or 4;
   			6:
   			Spon_messageblock[Spon_Pad_byteind] := Spon_messageblock[Spon_Pad_byteind] or 16#2;
   			7:
   				Spon_messageblock[Spon_Pad_byteind]:= Spon_messageblock[Spon_Pad_byteind] or 16#1;
   		End_case;
   	else
   		Spon_messageblock[Spon_Pad_byteind]:= 16#80;
   	end_if;
   
   	 while Spon_Pad_byteind<>Spon_R_SizeInBytes do
   
                   Spon_Pad_byteind:=Spon_Pad_byteind+1;
                   Spon_messageblock[Spon_Pad_byteind] := 0;
   	end_while;
   
END_ROUTINE

ROUTINE SPONGENT_Permute   (* structured text *)
   (*
   void Permute(hashState *state)
   {
   	bit16	i, j, IV, INV_IV;
   	for(i = 0; i < nRounds; i++){
   //Spon_State[1]:=0;
   		/* Add counter values */
   		state->value[0]			^= Spon_IV& 16#FF;
   		state->value[1]			^= (IV / 256) & 16#FF;
   		INV_IV	= retnuoCl(IV);
   		state->value[nSBox-1]	^= (INV_IV / 256) & 16#FF;;
   		state->value[nSBox-2]	^= INV_IV & 16#FF;
   		IV	= lCounter(IV);
   
   		/* sBoxLayer layer */
   		for ( j=0; j < nSBox; j++)
   			state->value[j] =  sBoxLayer[state->value[j]];
   		/* pLayer */
   		pLayer(state);
   	}
   }
   *)
   /*
   Case Spon_Ver Of
   		88808:
   			Spon_IV := 16#05;
   		8817688:
   			Spon_IV := 16#C6;
   		   1281288:	 Spon_IV:= 16#7A;
   		 128256128:	 Spon_IV:= 16#FB;
   		  16016016:	 Spon_IV:= 16#45;
   		  16016080:	 Spon_IV:= 16#01;
   		 160320160:	 Spon_IV:= 16#A7;
   		  22422416:	 Spon_IV:= 16#01;
   		 224224112:	 Spon_IV:= 16#52;
   		 224448224:	 Spon_IV:= 16#105;
   		  25625616:	 Spon_IV:= 16#9e;
   		 256256128:	 Spon_IV:= 16#fb;
   		 256512256:	 Spon_IV:= 16#015;
   End_case;
   */
   
   For Spon_Permute_i:=0 to Spon_nRounds-1 by 1 Do
   	Spon_State[0]:=Spon_State[0] XOR Spon_IV[Spon_Permute_i];
   	//Spon_State[1]:=Spon_State[1] XOR ((Spon_IV[Spon_Permute_i]/256) And 16#FF);
   
   	Spon_State[Spon_nSBox-1]:=Spon_State[Spon_nSBox-1] XOR ((Spon_INV_IV[Spon_Permute_i]/256) And 16#FF);
   	Spon_State[Spon_nSBox-2]:=Spon_State[Spon_nSBox-2] XOR ((Spon_INV_IV[Spon_Permute_i]) And 16#FF);
   
   
   
   		/*sLayer */
   	for Spon_Permute_j:=0 to Spon_nSBox-1 by 1 Do
   
   		Spon_Slayer_input:= Spon_State[Spon_Permute_j];
   		Spon_State[Spon_Permute_j]:=Spon_SBoxLayer[Spon_Slayer_input];
   
   	End_for;
   
   
   		/* pLayer */
   	jsr(SPONGENT_PLayer);
   
   End_For;
END_ROUTINE

ROUTINE SPONGENT_PLayer   (* structured text *)
   CASE Spon_Ver OF
   	 88808:
   		Spon_State_tmp[0].[0]:=Spon_State[0].[0];
   		Spon_State_tmp[2].[6]:=Spon_State[0].[1];
   		Spon_State_tmp[5].[4]:=Spon_State[0].[2];
   		Spon_State_tmp[8].[2]:=Spon_State[0].[3];
   		Spon_State_tmp[0].[1]:=Spon_State[0].[4];
   		Spon_State_tmp[2].[7]:=Spon_State[0].[5];
   		Spon_State_tmp[5].[5]:=Spon_State[0].[6];
   		Spon_State_tmp[8].[3]:=Spon_State[0].[7];
   		Spon_State_tmp[0].[2]:=Spon_State[1].[0];
   		Spon_State_tmp[3].[0]:=Spon_State[1].[1];
   		Spon_State_tmp[5].[6]:=Spon_State[1].[2];
   		Spon_State_tmp[8].[4]:=Spon_State[1].[3];
   		Spon_State_tmp[0].[3]:=Spon_State[1].[4];
   		Spon_State_tmp[3].[1]:=Spon_State[1].[5];
   		Spon_State_tmp[5].[7]:=Spon_State[1].[6];
   		Spon_State_tmp[8].[5]:=Spon_State[1].[7];
   		Spon_State_tmp[0].[4]:=Spon_State[2].[0];
   		Spon_State_tmp[3].[2]:=Spon_State[2].[1];
   		Spon_State_tmp[6].[0]:=Spon_State[2].[2];
   		Spon_State_tmp[8].[6]:=Spon_State[2].[3];
   		Spon_State_tmp[0].[5]:=Spon_State[2].[4];
   		Spon_State_tmp[3].[3]:=Spon_State[2].[5];
   		Spon_State_tmp[6].[1]:=Spon_State[2].[6];
   		Spon_State_tmp[8].[7]:=Spon_State[2].[7];
   		Spon_State_tmp[0].[6]:=Spon_State[3].[0];
   		Spon_State_tmp[3].[4]:=Spon_State[3].[1];
   		Spon_State_tmp[6].[2]:=Spon_State[3].[2];
   		Spon_State_tmp[9].[0]:=Spon_State[3].[3];
   		Spon_State_tmp[0].[7]:=Spon_State[3].[4];
   		Spon_State_tmp[3].[5]:=Spon_State[3].[5];
   		Spon_State_tmp[6].[3]:=Spon_State[3].[6];
   		Spon_State_tmp[9].[1]:=Spon_State[3].[7];
   		Spon_State_tmp[1].[0]:=Spon_State[4].[0];
   		Spon_State_tmp[3].[6]:=Spon_State[4].[1];
   		Spon_State_tmp[6].[4]:=Spon_State[4].[2];
   		Spon_State_tmp[9].[2]:=Spon_State[4].[3];
   		Spon_State_tmp[1].[1]:=Spon_State[4].[4];
   		Spon_State_tmp[3].[7]:=Spon_State[4].[5];
   		Spon_State_tmp[6].[5]:=Spon_State[4].[6];
   		Spon_State_tmp[9].[3]:=Spon_State[4].[7];
   		Spon_State_tmp[1].[2]:=Spon_State[5].[0];
   		Spon_State_tmp[4].[0]:=Spon_State[5].[1];
   		Spon_State_tmp[6].[6]:=Spon_State[5].[2];
   		Spon_State_tmp[9].[4]:=Spon_State[5].[3];
   		Spon_State_tmp[1].[3]:=Spon_State[5].[4];
   		Spon_State_tmp[4].[1]:=Spon_State[5].[5];
   		Spon_State_tmp[6].[7]:=Spon_State[5].[6];
   		Spon_State_tmp[9].[5]:=Spon_State[5].[7];
   		Spon_State_tmp[1].[4]:=Spon_State[6].[0];
   		Spon_State_tmp[4].[2]:=Spon_State[6].[1];
   		Spon_State_tmp[7].[0]:=Spon_State[6].[2];
   		Spon_State_tmp[9].[6]:=Spon_State[6].[3];
   		Spon_State_tmp[1].[5]:=Spon_State[6].[4];
   		Spon_State_tmp[4].[3]:=Spon_State[6].[5];
   		Spon_State_tmp[7].[1]:=Spon_State[6].[6];
   		Spon_State_tmp[9].[7]:=Spon_State[6].[7];
   		Spon_State_tmp[1].[6]:=Spon_State[7].[0];
   		Spon_State_tmp[4].[4]:=Spon_State[7].[1];
   		Spon_State_tmp[7].[2]:=Spon_State[7].[2];
   		Spon_State_tmp[10].[0]:=Spon_State[7].[3];
   		Spon_State_tmp[1].[7]:=Spon_State[7].[4];
   		Spon_State_tmp[4].[5]:=Spon_State[7].[5];
   		Spon_State_tmp[7].[3]:=Spon_State[7].[6];
   		Spon_State_tmp[10].[1]:=Spon_State[7].[7];
   		Spon_State_tmp[2].[0]:=Spon_State[8].[0];
   		Spon_State_tmp[4].[6]:=Spon_State[8].[1];
   		Spon_State_tmp[7].[4]:=Spon_State[8].[2];
   		Spon_State_tmp[10].[2]:=Spon_State[8].[3];
   		Spon_State_tmp[2].[1]:=Spon_State[8].[4];
   		Spon_State_tmp[4].[7]:=Spon_State[8].[5];
   		Spon_State_tmp[7].[5]:=Spon_State[8].[6];
   		Spon_State_tmp[10].[3]:=Spon_State[8].[7];
   		Spon_State_tmp[2].[2]:=Spon_State[9].[0];
   		Spon_State_tmp[5].[0]:=Spon_State[9].[1];
   		Spon_State_tmp[7].[6]:=Spon_State[9].[2];
   		Spon_State_tmp[10].[4]:=Spon_State[9].[3];
   		Spon_State_tmp[2].[3]:=Spon_State[9].[4];
   		Spon_State_tmp[5].[1]:=Spon_State[9].[5];
   		Spon_State_tmp[7].[7]:=Spon_State[9].[6];
   		Spon_State_tmp[10].[5]:=Spon_State[9].[7];
   		Spon_State_tmp[2].[4]:=Spon_State[10].[0];
   		Spon_State_tmp[5].[2]:=Spon_State[10].[1];
   		Spon_State_tmp[8].[0]:=Spon_State[10].[2];
   		Spon_State_tmp[10].[6]:=Spon_State[10].[3];
   		Spon_State_tmp[2].[5]:=Spon_State[10].[4];
   		Spon_State_tmp[5].[3]:=Spon_State[10].[5];
   		Spon_State_tmp[8].[1]:=Spon_State[10].[6];
   		Spon_State_tmp[10].[7]:=Spon_State[10].[7];
   	 8817688:
   		Spon_State_tmp[0].[0]:=Spon_State[0].[0];
   		Spon_State_tmp[8].[2]:=Spon_State[0].[1];
   		Spon_State_tmp[16].[4]:=Spon_State[0].[2];
   		Spon_State_tmp[24].[6]:=Spon_State[0].[3];
   		Spon_State_tmp[0].[1]:=Spon_State[0].[4];
   		Spon_State_tmp[8].[3]:=Spon_State[0].[5];
   		Spon_State_tmp[16].[5]:=Spon_State[0].[6];
   		Spon_State_tmp[24].[7]:=Spon_State[0].[7];
   		Spon_State_tmp[0].[2]:=Spon_State[1].[0];
   		Spon_State_tmp[8].[4]:=Spon_State[1].[1];
   		Spon_State_tmp[16].[6]:=Spon_State[1].[2];
   		Spon_State_tmp[25].[0]:=Spon_State[1].[3];
   		Spon_State_tmp[0].[3]:=Spon_State[1].[4];
   		Spon_State_tmp[8].[5]:=Spon_State[1].[5];
   		Spon_State_tmp[16].[7]:=Spon_State[1].[6];
   		Spon_State_tmp[25].[1]:=Spon_State[1].[7];
   		Spon_State_tmp[0].[4]:=Spon_State[2].[0];
   		Spon_State_tmp[8].[6]:=Spon_State[2].[1];
   		Spon_State_tmp[17].[0]:=Spon_State[2].[2];
   		Spon_State_tmp[25].[2]:=Spon_State[2].[3];
   		Spon_State_tmp[0].[5]:=Spon_State[2].[4];
   		Spon_State_tmp[8].[7]:=Spon_State[2].[5];
   		Spon_State_tmp[17].[1]:=Spon_State[2].[6];
   		Spon_State_tmp[25].[3]:=Spon_State[2].[7];
   		Spon_State_tmp[0].[6]:=Spon_State[3].[0];
   		Spon_State_tmp[9].[0]:=Spon_State[3].[1];
   		Spon_State_tmp[17].[2]:=Spon_State[3].[2];
   		Spon_State_tmp[25].[4]:=Spon_State[3].[3];
   		Spon_State_tmp[0].[7]:=Spon_State[3].[4];
   		Spon_State_tmp[9].[1]:=Spon_State[3].[5];
   		Spon_State_tmp[17].[3]:=Spon_State[3].[6];
   		Spon_State_tmp[25].[5]:=Spon_State[3].[7];
   		Spon_State_tmp[1].[0]:=Spon_State[4].[0];
   		Spon_State_tmp[9].[2]:=Spon_State[4].[1];
   		Spon_State_tmp[17].[4]:=Spon_State[4].[2];
   		Spon_State_tmp[25].[6]:=Spon_State[4].[3];
   		Spon_State_tmp[1].[1]:=Spon_State[4].[4];
   		Spon_State_tmp[9].[3]:=Spon_State[4].[5];
   		Spon_State_tmp[17].[5]:=Spon_State[4].[6];
   		Spon_State_tmp[25].[7]:=Spon_State[4].[7];
   		Spon_State_tmp[1].[2]:=Spon_State[5].[0];
   		Spon_State_tmp[9].[4]:=Spon_State[5].[1];
   		Spon_State_tmp[17].[6]:=Spon_State[5].[2];
   		Spon_State_tmp[26].[0]:=Spon_State[5].[3];
   		Spon_State_tmp[1].[3]:=Spon_State[5].[4];
   		Spon_State_tmp[9].[5]:=Spon_State[5].[5];
   		Spon_State_tmp[17].[7]:=Spon_State[5].[6];
   		Spon_State_tmp[26].[1]:=Spon_State[5].[7];
   		Spon_State_tmp[1].[4]:=Spon_State[6].[0];
   		Spon_State_tmp[9].[6]:=Spon_State[6].[1];
   		Spon_State_tmp[18].[0]:=Spon_State[6].[2];
   		Spon_State_tmp[26].[2]:=Spon_State[6].[3];
   		Spon_State_tmp[1].[5]:=Spon_State[6].[4];
   		Spon_State_tmp[9].[7]:=Spon_State[6].[5];
   		Spon_State_tmp[18].[1]:=Spon_State[6].[6];
   		Spon_State_tmp[26].[3]:=Spon_State[6].[7];
   		Spon_State_tmp[1].[6]:=Spon_State[7].[0];
   		Spon_State_tmp[10].[0]:=Spon_State[7].[1];
   		Spon_State_tmp[18].[2]:=Spon_State[7].[2];
   		Spon_State_tmp[26].[4]:=Spon_State[7].[3];
   		Spon_State_tmp[1].[7]:=Spon_State[7].[4];
   		Spon_State_tmp[10].[1]:=Spon_State[7].[5];
   		Spon_State_tmp[18].[3]:=Spon_State[7].[6];
   		Spon_State_tmp[26].[5]:=Spon_State[7].[7];
   		Spon_State_tmp[2].[0]:=Spon_State[8].[0];
   		Spon_State_tmp[10].[2]:=Spon_State[8].[1];
   		Spon_State_tmp[18].[4]:=Spon_State[8].[2];
   		Spon_State_tmp[26].[6]:=Spon_State[8].[3];
   		Spon_State_tmp[2].[1]:=Spon_State[8].[4];
   		Spon_State_tmp[10].[3]:=Spon_State[8].[5];
   		Spon_State_tmp[18].[5]:=Spon_State[8].[6];
   		Spon_State_tmp[26].[7]:=Spon_State[8].[7];
   		Spon_State_tmp[2].[2]:=Spon_State[9].[0];
   		Spon_State_tmp[10].[4]:=Spon_State[9].[1];
   		Spon_State_tmp[18].[6]:=Spon_State[9].[2];
   		Spon_State_tmp[27].[0]:=Spon_State[9].[3];
   		Spon_State_tmp[2].[3]:=Spon_State[9].[4];
   		Spon_State_tmp[10].[5]:=Spon_State[9].[5];
   		Spon_State_tmp[18].[7]:=Spon_State[9].[6];
   		Spon_State_tmp[27].[1]:=Spon_State[9].[7];
   		Spon_State_tmp[2].[4]:=Spon_State[10].[0];
   		Spon_State_tmp[10].[6]:=Spon_State[10].[1];
   		Spon_State_tmp[19].[0]:=Spon_State[10].[2];
   		Spon_State_tmp[27].[2]:=Spon_State[10].[3];
   		Spon_State_tmp[2].[5]:=Spon_State[10].[4];
   		Spon_State_tmp[10].[7]:=Spon_State[10].[5];
   		Spon_State_tmp[19].[1]:=Spon_State[10].[6];
   		Spon_State_tmp[27].[3]:=Spon_State[10].[7];
   		Spon_State_tmp[2].[6]:=Spon_State[11].[0];
   		Spon_State_tmp[11].[0]:=Spon_State[11].[1];
   		Spon_State_tmp[19].[2]:=Spon_State[11].[2];
   		Spon_State_tmp[27].[4]:=Spon_State[11].[3];
   		Spon_State_tmp[2].[7]:=Spon_State[11].[4];
   		Spon_State_tmp[11].[1]:=Spon_State[11].[5];
   		Spon_State_tmp[19].[3]:=Spon_State[11].[6];
   		Spon_State_tmp[27].[5]:=Spon_State[11].[7];
   		Spon_State_tmp[3].[0]:=Spon_State[12].[0];
   		Spon_State_tmp[11].[2]:=Spon_State[12].[1];
   		Spon_State_tmp[19].[4]:=Spon_State[12].[2];
   		Spon_State_tmp[27].[6]:=Spon_State[12].[3];
   		Spon_State_tmp[3].[1]:=Spon_State[12].[4];
   		Spon_State_tmp[11].[3]:=Spon_State[12].[5];
   		Spon_State_tmp[19].[5]:=Spon_State[12].[6];
   		Spon_State_tmp[27].[7]:=Spon_State[12].[7];
   		Spon_State_tmp[3].[2]:=Spon_State[13].[0];
   		Spon_State_tmp[11].[4]:=Spon_State[13].[1];
   		Spon_State_tmp[19].[6]:=Spon_State[13].[2];
   		Spon_State_tmp[28].[0]:=Spon_State[13].[3];
   		Spon_State_tmp[3].[3]:=Spon_State[13].[4];
   		Spon_State_tmp[11].[5]:=Spon_State[13].[5];
   		Spon_State_tmp[19].[7]:=Spon_State[13].[6];
   		Spon_State_tmp[28].[1]:=Spon_State[13].[7];
   		Spon_State_tmp[3].[4]:=Spon_State[14].[0];
   		Spon_State_tmp[11].[6]:=Spon_State[14].[1];
   		Spon_State_tmp[20].[0]:=Spon_State[14].[2];
   		Spon_State_tmp[28].[2]:=Spon_State[14].[3];
   		Spon_State_tmp[3].[5]:=Spon_State[14].[4];
   		Spon_State_tmp[11].[7]:=Spon_State[14].[5];
   		Spon_State_tmp[20].[1]:=Spon_State[14].[6];
   		Spon_State_tmp[28].[3]:=Spon_State[14].[7];
   		Spon_State_tmp[3].[6]:=Spon_State[15].[0];
   		Spon_State_tmp[12].[0]:=Spon_State[15].[1];
   		Spon_State_tmp[20].[2]:=Spon_State[15].[2];
   		Spon_State_tmp[28].[4]:=Spon_State[15].[3];
   		Spon_State_tmp[3].[7]:=Spon_State[15].[4];
   		Spon_State_tmp[12].[1]:=Spon_State[15].[5];
   		Spon_State_tmp[20].[3]:=Spon_State[15].[6];
   		Spon_State_tmp[28].[5]:=Spon_State[15].[7];
   		Spon_State_tmp[4].[0]:=Spon_State[16].[0];
   		Spon_State_tmp[12].[2]:=Spon_State[16].[1];
   		Spon_State_tmp[20].[4]:=Spon_State[16].[2];
   		Spon_State_tmp[28].[6]:=Spon_State[16].[3];
   		Spon_State_tmp[4].[1]:=Spon_State[16].[4];
   		Spon_State_tmp[12].[3]:=Spon_State[16].[5];
   		Spon_State_tmp[20].[5]:=Spon_State[16].[6];
   		Spon_State_tmp[28].[7]:=Spon_State[16].[7];
   		Spon_State_tmp[4].[2]:=Spon_State[17].[0];
   		Spon_State_tmp[12].[4]:=Spon_State[17].[1];
   		Spon_State_tmp[20].[6]:=Spon_State[17].[2];
   		Spon_State_tmp[29].[0]:=Spon_State[17].[3];
   		Spon_State_tmp[4].[3]:=Spon_State[17].[4];
   		Spon_State_tmp[12].[5]:=Spon_State[17].[5];
   		Spon_State_tmp[20].[7]:=Spon_State[17].[6];
   		Spon_State_tmp[29].[1]:=Spon_State[17].[7];
   		Spon_State_tmp[4].[4]:=Spon_State[18].[0];
   		Spon_State_tmp[12].[6]:=Spon_State[18].[1];
   		Spon_State_tmp[21].[0]:=Spon_State[18].[2];
   		Spon_State_tmp[29].[2]:=Spon_State[18].[3];
   		Spon_State_tmp[4].[5]:=Spon_State[18].[4];
   		Spon_State_tmp[12].[7]:=Spon_State[18].[5];
   		Spon_State_tmp[21].[1]:=Spon_State[18].[6];
   		Spon_State_tmp[29].[3]:=Spon_State[18].[7];
   		Spon_State_tmp[4].[6]:=Spon_State[19].[0];
   		Spon_State_tmp[13].[0]:=Spon_State[19].[1];
   		Spon_State_tmp[21].[2]:=Spon_State[19].[2];
   		Spon_State_tmp[29].[4]:=Spon_State[19].[3];
   		Spon_State_tmp[4].[7]:=Spon_State[19].[4];
   		Spon_State_tmp[13].[1]:=Spon_State[19].[5];
   		Spon_State_tmp[21].[3]:=Spon_State[19].[6];
   		Spon_State_tmp[29].[5]:=Spon_State[19].[7];
   		Spon_State_tmp[5].[0]:=Spon_State[20].[0];
   		Spon_State_tmp[13].[2]:=Spon_State[20].[1];
   		Spon_State_tmp[21].[4]:=Spon_State[20].[2];
   		Spon_State_tmp[29].[6]:=Spon_State[20].[3];
   		Spon_State_tmp[5].[1]:=Spon_State[20].[4];
   		Spon_State_tmp[13].[3]:=Spon_State[20].[5];
   		Spon_State_tmp[21].[5]:=Spon_State[20].[6];
   		Spon_State_tmp[29].[7]:=Spon_State[20].[7];
   		Spon_State_tmp[5].[2]:=Spon_State[21].[0];
   		Spon_State_tmp[13].[4]:=Spon_State[21].[1];
   		Spon_State_tmp[21].[6]:=Spon_State[21].[2];
   		Spon_State_tmp[30].[0]:=Spon_State[21].[3];
   		Spon_State_tmp[5].[3]:=Spon_State[21].[4];
   		Spon_State_tmp[13].[5]:=Spon_State[21].[5];
   		Spon_State_tmp[21].[7]:=Spon_State[21].[6];
   		Spon_State_tmp[30].[1]:=Spon_State[21].[7];
   		Spon_State_tmp[5].[4]:=Spon_State[22].[0];
   		Spon_State_tmp[13].[6]:=Spon_State[22].[1];
   		Spon_State_tmp[22].[0]:=Spon_State[22].[2];
   		Spon_State_tmp[30].[2]:=Spon_State[22].[3];
   		Spon_State_tmp[5].[5]:=Spon_State[22].[4];
   		Spon_State_tmp[13].[7]:=Spon_State[22].[5];
   		Spon_State_tmp[22].[1]:=Spon_State[22].[6];
   		Spon_State_tmp[30].[3]:=Spon_State[22].[7];
   		Spon_State_tmp[5].[6]:=Spon_State[23].[0];
   		Spon_State_tmp[14].[0]:=Spon_State[23].[1];
   		Spon_State_tmp[22].[2]:=Spon_State[23].[2];
   		Spon_State_tmp[30].[4]:=Spon_State[23].[3];
   		Spon_State_tmp[5].[7]:=Spon_State[23].[4];
   		Spon_State_tmp[14].[1]:=Spon_State[23].[5];
   		Spon_State_tmp[22].[3]:=Spon_State[23].[6];
   		Spon_State_tmp[30].[5]:=Spon_State[23].[7];
   		Spon_State_tmp[6].[0]:=Spon_State[24].[0];
   		Spon_State_tmp[14].[2]:=Spon_State[24].[1];
   		Spon_State_tmp[22].[4]:=Spon_State[24].[2];
   		Spon_State_tmp[30].[6]:=Spon_State[24].[3];
   		Spon_State_tmp[6].[1]:=Spon_State[24].[4];
   		Spon_State_tmp[14].[3]:=Spon_State[24].[5];
   		Spon_State_tmp[22].[5]:=Spon_State[24].[6];
   		Spon_State_tmp[30].[7]:=Spon_State[24].[7];
   		Spon_State_tmp[6].[2]:=Spon_State[25].[0];
   		Spon_State_tmp[14].[4]:=Spon_State[25].[1];
   		Spon_State_tmp[22].[6]:=Spon_State[25].[2];
   		Spon_State_tmp[31].[0]:=Spon_State[25].[3];
   		Spon_State_tmp[6].[3]:=Spon_State[25].[4];
   		Spon_State_tmp[14].[5]:=Spon_State[25].[5];
   		Spon_State_tmp[22].[7]:=Spon_State[25].[6];
   		Spon_State_tmp[31].[1]:=Spon_State[25].[7];
   		Spon_State_tmp[6].[4]:=Spon_State[26].[0];
   		Spon_State_tmp[14].[6]:=Spon_State[26].[1];
   		Spon_State_tmp[23].[0]:=Spon_State[26].[2];
   		Spon_State_tmp[31].[2]:=Spon_State[26].[3];
   		Spon_State_tmp[6].[5]:=Spon_State[26].[4];
   		Spon_State_tmp[14].[7]:=Spon_State[26].[5];
   		Spon_State_tmp[23].[1]:=Spon_State[26].[6];
   		Spon_State_tmp[31].[3]:=Spon_State[26].[7];
   		Spon_State_tmp[6].[6]:=Spon_State[27].[0];
   		Spon_State_tmp[15].[0]:=Spon_State[27].[1];
   		Spon_State_tmp[23].[2]:=Spon_State[27].[2];
   		Spon_State_tmp[31].[4]:=Spon_State[27].[3];
   		Spon_State_tmp[6].[7]:=Spon_State[27].[4];
   		Spon_State_tmp[15].[1]:=Spon_State[27].[5];
   		Spon_State_tmp[23].[3]:=Spon_State[27].[6];
   		Spon_State_tmp[31].[5]:=Spon_State[27].[7];
   		Spon_State_tmp[7].[0]:=Spon_State[28].[0];
   		Spon_State_tmp[15].[2]:=Spon_State[28].[1];
   		Spon_State_tmp[23].[4]:=Spon_State[28].[2];
   		Spon_State_tmp[31].[6]:=Spon_State[28].[3];
   		Spon_State_tmp[7].[1]:=Spon_State[28].[4];
   		Spon_State_tmp[15].[3]:=Spon_State[28].[5];
   		Spon_State_tmp[23].[5]:=Spon_State[28].[6];
   		Spon_State_tmp[31].[7]:=Spon_State[28].[7];
   		Spon_State_tmp[7].[2]:=Spon_State[29].[0];
   		Spon_State_tmp[15].[4]:=Spon_State[29].[1];
   		Spon_State_tmp[23].[6]:=Spon_State[29].[2];
   		Spon_State_tmp[32].[0]:=Spon_State[29].[3];
   		Spon_State_tmp[7].[3]:=Spon_State[29].[4];
   		Spon_State_tmp[15].[5]:=Spon_State[29].[5];
   		Spon_State_tmp[23].[7]:=Spon_State[29].[6];
   		Spon_State_tmp[32].[1]:=Spon_State[29].[7];
   		Spon_State_tmp[7].[4]:=Spon_State[30].[0];
   		Spon_State_tmp[15].[6]:=Spon_State[30].[1];
   		Spon_State_tmp[24].[0]:=Spon_State[30].[2];
   		Spon_State_tmp[32].[2]:=Spon_State[30].[3];
   		Spon_State_tmp[7].[5]:=Spon_State[30].[4];
   		Spon_State_tmp[15].[7]:=Spon_State[30].[5];
   		Spon_State_tmp[24].[1]:=Spon_State[30].[6];
   		Spon_State_tmp[32].[3]:=Spon_State[30].[7];
   		Spon_State_tmp[7].[6]:=Spon_State[31].[0];
   		Spon_State_tmp[16].[0]:=Spon_State[31].[1];
   		Spon_State_tmp[24].[2]:=Spon_State[31].[2];
   		Spon_State_tmp[32].[4]:=Spon_State[31].[3];
   		Spon_State_tmp[7].[7]:=Spon_State[31].[4];
   		Spon_State_tmp[16].[1]:=Spon_State[31].[5];
   		Spon_State_tmp[24].[3]:=Spon_State[31].[6];
   		Spon_State_tmp[32].[5]:=Spon_State[31].[7];
   		Spon_State_tmp[8].[0]:=Spon_State[32].[0];
   		Spon_State_tmp[16].[2]:=Spon_State[32].[1];
   		Spon_State_tmp[24].[4]:=Spon_State[32].[2];
   		Spon_State_tmp[32].[6]:=Spon_State[32].[3];
   		Spon_State_tmp[8].[1]:=Spon_State[32].[4];
   		Spon_State_tmp[16].[3]:=Spon_State[32].[5];
   		Spon_State_tmp[24].[5]:=Spon_State[32].[6];
   		Spon_State_tmp[32].[7]:=Spon_State[32].[7];
   	 1281288:
   		Spon_State_tmp[0].[0]:=Spon_State[0].[0];
   		Spon_State_tmp[4].[2]:=Spon_State[0].[1];
   		Spon_State_tmp[8].[4]:=Spon_State[0].[2];
   		Spon_State_tmp[12].[6]:=Spon_State[0].[3];
   		Spon_State_tmp[0].[1]:=Spon_State[0].[4];
   		Spon_State_tmp[4].[3]:=Spon_State[0].[5];
   		Spon_State_tmp[8].[5]:=Spon_State[0].[6];
   		Spon_State_tmp[12].[7]:=Spon_State[0].[7];
   		Spon_State_tmp[0].[2]:=Spon_State[1].[0];
   		Spon_State_tmp[4].[4]:=Spon_State[1].[1];
   		Spon_State_tmp[8].[6]:=Spon_State[1].[2];
   		Spon_State_tmp[13].[0]:=Spon_State[1].[3];
   		Spon_State_tmp[0].[3]:=Spon_State[1].[4];
   		Spon_State_tmp[4].[5]:=Spon_State[1].[5];
   		Spon_State_tmp[8].[7]:=Spon_State[1].[6];
   		Spon_State_tmp[13].[1]:=Spon_State[1].[7];
   		Spon_State_tmp[0].[4]:=Spon_State[2].[0];
   		Spon_State_tmp[4].[6]:=Spon_State[2].[1];
   		Spon_State_tmp[9].[0]:=Spon_State[2].[2];
   		Spon_State_tmp[13].[2]:=Spon_State[2].[3];
   		Spon_State_tmp[0].[5]:=Spon_State[2].[4];
   		Spon_State_tmp[4].[7]:=Spon_State[2].[5];
   		Spon_State_tmp[9].[1]:=Spon_State[2].[6];
   		Spon_State_tmp[13].[3]:=Spon_State[2].[7];
   		Spon_State_tmp[0].[6]:=Spon_State[3].[0];
   		Spon_State_tmp[5].[0]:=Spon_State[3].[1];
   		Spon_State_tmp[9].[2]:=Spon_State[3].[2];
   		Spon_State_tmp[13].[4]:=Spon_State[3].[3];
   		Spon_State_tmp[0].[7]:=Spon_State[3].[4];
   		Spon_State_tmp[5].[1]:=Spon_State[3].[5];
   		Spon_State_tmp[9].[3]:=Spon_State[3].[6];
   		Spon_State_tmp[13].[5]:=Spon_State[3].[7];
   		Spon_State_tmp[1].[0]:=Spon_State[4].[0];
   		Spon_State_tmp[5].[2]:=Spon_State[4].[1];
   		Spon_State_tmp[9].[4]:=Spon_State[4].[2];
   		Spon_State_tmp[13].[6]:=Spon_State[4].[3];
   		Spon_State_tmp[1].[1]:=Spon_State[4].[4];
   		Spon_State_tmp[5].[3]:=Spon_State[4].[5];
   		Spon_State_tmp[9].[5]:=Spon_State[4].[6];
   		Spon_State_tmp[13].[7]:=Spon_State[4].[7];
   		Spon_State_tmp[1].[2]:=Spon_State[5].[0];
   		Spon_State_tmp[5].[4]:=Spon_State[5].[1];
   		Spon_State_tmp[9].[6]:=Spon_State[5].[2];
   		Spon_State_tmp[14].[0]:=Spon_State[5].[3];
   		Spon_State_tmp[1].[3]:=Spon_State[5].[4];
   		Spon_State_tmp[5].[5]:=Spon_State[5].[5];
   		Spon_State_tmp[9].[7]:=Spon_State[5].[6];
   		Spon_State_tmp[14].[1]:=Spon_State[5].[7];
   		Spon_State_tmp[1].[4]:=Spon_State[6].[0];
   		Spon_State_tmp[5].[6]:=Spon_State[6].[1];
   		Spon_State_tmp[10].[0]:=Spon_State[6].[2];
   		Spon_State_tmp[14].[2]:=Spon_State[6].[3];
   		Spon_State_tmp[1].[5]:=Spon_State[6].[4];
   		Spon_State_tmp[5].[7]:=Spon_State[6].[5];
   		Spon_State_tmp[10].[1]:=Spon_State[6].[6];
   		Spon_State_tmp[14].[3]:=Spon_State[6].[7];
   		Spon_State_tmp[1].[6]:=Spon_State[7].[0];
   		Spon_State_tmp[6].[0]:=Spon_State[7].[1];
   		Spon_State_tmp[10].[2]:=Spon_State[7].[2];
   		Spon_State_tmp[14].[4]:=Spon_State[7].[3];
   		Spon_State_tmp[1].[7]:=Spon_State[7].[4];
   		Spon_State_tmp[6].[1]:=Spon_State[7].[5];
   		Spon_State_tmp[10].[3]:=Spon_State[7].[6];
   		Spon_State_tmp[14].[5]:=Spon_State[7].[7];
   		Spon_State_tmp[2].[0]:=Spon_State[8].[0];
   		Spon_State_tmp[6].[2]:=Spon_State[8].[1];
   		Spon_State_tmp[10].[4]:=Spon_State[8].[2];
   		Spon_State_tmp[14].[6]:=Spon_State[8].[3];
   		Spon_State_tmp[2].[1]:=Spon_State[8].[4];
   		Spon_State_tmp[6].[3]:=Spon_State[8].[5];
   		Spon_State_tmp[10].[5]:=Spon_State[8].[6];
   		Spon_State_tmp[14].[7]:=Spon_State[8].[7];
   		Spon_State_tmp[2].[2]:=Spon_State[9].[0];
   		Spon_State_tmp[6].[4]:=Spon_State[9].[1];
   		Spon_State_tmp[10].[6]:=Spon_State[9].[2];
   		Spon_State_tmp[15].[0]:=Spon_State[9].[3];
   		Spon_State_tmp[2].[3]:=Spon_State[9].[4];
   		Spon_State_tmp[6].[5]:=Spon_State[9].[5];
   		Spon_State_tmp[10].[7]:=Spon_State[9].[6];
   		Spon_State_tmp[15].[1]:=Spon_State[9].[7];
   		Spon_State_tmp[2].[4]:=Spon_State[10].[0];
   		Spon_State_tmp[6].[6]:=Spon_State[10].[1];
   		Spon_State_tmp[11].[0]:=Spon_State[10].[2];
   		Spon_State_tmp[15].[2]:=Spon_State[10].[3];
   		Spon_State_tmp[2].[5]:=Spon_State[10].[4];
   		Spon_State_tmp[6].[7]:=Spon_State[10].[5];
   		Spon_State_tmp[11].[1]:=Spon_State[10].[6];
   		Spon_State_tmp[15].[3]:=Spon_State[10].[7];
   		Spon_State_tmp[2].[6]:=Spon_State[11].[0];
   		Spon_State_tmp[7].[0]:=Spon_State[11].[1];
   		Spon_State_tmp[11].[2]:=Spon_State[11].[2];
   		Spon_State_tmp[15].[4]:=Spon_State[11].[3];
   		Spon_State_tmp[2].[7]:=Spon_State[11].[4];
   		Spon_State_tmp[7].[1]:=Spon_State[11].[5];
   		Spon_State_tmp[11].[3]:=Spon_State[11].[6];
   		Spon_State_tmp[15].[5]:=Spon_State[11].[7];
   		Spon_State_tmp[3].[0]:=Spon_State[12].[0];
   		Spon_State_tmp[7].[2]:=Spon_State[12].[1];
   		Spon_State_tmp[11].[4]:=Spon_State[12].[2];
   		Spon_State_tmp[15].[6]:=Spon_State[12].[3];
   		Spon_State_tmp[3].[1]:=Spon_State[12].[4];
   		Spon_State_tmp[7].[3]:=Spon_State[12].[5];
   		Spon_State_tmp[11].[5]:=Spon_State[12].[6];
   		Spon_State_tmp[15].[7]:=Spon_State[12].[7];
   		Spon_State_tmp[3].[2]:=Spon_State[13].[0];
   		Spon_State_tmp[7].[4]:=Spon_State[13].[1];
   		Spon_State_tmp[11].[6]:=Spon_State[13].[2];
   		Spon_State_tmp[16].[0]:=Spon_State[13].[3];
   		Spon_State_tmp[3].[3]:=Spon_State[13].[4];
   		Spon_State_tmp[7].[5]:=Spon_State[13].[5];
   		Spon_State_tmp[11].[7]:=Spon_State[13].[6];
   		Spon_State_tmp[16].[1]:=Spon_State[13].[7];
   		Spon_State_tmp[3].[4]:=Spon_State[14].[0];
   		Spon_State_tmp[7].[6]:=Spon_State[14].[1];
   		Spon_State_tmp[12].[0]:=Spon_State[14].[2];
   		Spon_State_tmp[16].[2]:=Spon_State[14].[3];
   		Spon_State_tmp[3].[5]:=Spon_State[14].[4];
   		Spon_State_tmp[7].[7]:=Spon_State[14].[5];
   		Spon_State_tmp[12].[1]:=Spon_State[14].[6];
   		Spon_State_tmp[16].[3]:=Spon_State[14].[7];
   		Spon_State_tmp[3].[6]:=Spon_State[15].[0];
   		Spon_State_tmp[8].[0]:=Spon_State[15].[1];
   		Spon_State_tmp[12].[2]:=Spon_State[15].[2];
   		Spon_State_tmp[16].[4]:=Spon_State[15].[3];
   		Spon_State_tmp[3].[7]:=Spon_State[15].[4];
   		Spon_State_tmp[8].[1]:=Spon_State[15].[5];
   		Spon_State_tmp[12].[3]:=Spon_State[15].[6];
   		Spon_State_tmp[16].[5]:=Spon_State[15].[7];
   		Spon_State_tmp[4].[0]:=Spon_State[16].[0];
   		Spon_State_tmp[8].[2]:=Spon_State[16].[1];
   		Spon_State_tmp[12].[4]:=Spon_State[16].[2];
   		Spon_State_tmp[16].[6]:=Spon_State[16].[3];
   		Spon_State_tmp[4].[1]:=Spon_State[16].[4];
   		Spon_State_tmp[8].[3]:=Spon_State[16].[5];
   		Spon_State_tmp[12].[5]:=Spon_State[16].[6];
   		Spon_State_tmp[16].[7]:=Spon_State[16].[7];
   End_CASE;
   
   
   For Spon_Player_i:=0 to Spon_nSBox-1 by 1 Do
   	Spon_State[Spon_Player_i]:=Spon_State_tmp[Spon_Player_i];
   End_For;
   
   
END_ROUTINE

ROUTINE SPONGENT_Squeeze   (* structured text *)
   (*
   HashReturn Squeeze(hashState *state)
   {
   	memcpy(state->messageblock, state->value, R_SizeInBytes);
   
   	Permute(state);
   
   	return SUCCESS;
   }
   
   *)
   
   For Spon_Squeeze_i:=0 to Spon_R_SizeInBytes-1 by 1 Do
   
   	Spon_messageblock[Spon_Squeeze_i]:= Spon_State[Spon_Squeeze_i];
   End_for;
   
   	jsr(SPONGENT_Permute);
   
END_ROUTINE

ROUTINE SPONGENT_Test   (* structured text *)
   
   
   if S:FS Then
   	Spon_Ver:=8817688;
   
   	Spon_MsgBitLen:=216;
   	for Test_i:=0 to Spon_MsgBitLen/8-1 by 1 do
   		Spon_Message[Test_i]:=48;
   	end_for;
   
   	for Test_i:=0 to Spon_DIGESTSIZE-1 by 1 do
   		Spon_Digest[Test_i]:=0;
   	end_for;
   
   //Jsr(SPONGENT_Init);
   
   
   
   end_if;
   
   Spon_MsgBitLen:=216;
   JSR(SPONGENT);
END_ROUTINE
END_PROGRAM
